# EPICS substitutions: EX2/scr/neurons_old.substitutions
file network.template {
	pattern { name, name-next, in1, w1, in2, w2, in3, w3, in4, w4}

		{ "11", "12-sum", "01", "01-11", "11", "11-11", "12", "12-11", "13", "13-11" }
		{ "12", "13-sum", "01", "01-12", "11", "11-12", "12", "12-12", "13", "13-12" }
		{ "13", "11-ac", "01", "01-13", "11", "11-13", "12", "12-13", "13", "13-13" }

		{ "21", "22-sum", "11", "11-21", "12", "12-21", "13", "13-21", "null", "null" }
		{ "22", "23-sum", "11", "11-22", "12", "12-22", "13", "13-22", "null", "null" }
		{ "23", "21-ac", "11", "11-23", "12", "12-23", "13", "13-23", "null", "null" }
}

file ac.template {
	pattern { name, name-next }
		{ "11", "12-ac" }
		{ "12", "13-ac" }
		{ "13", "21-sum" }

		{ "21", "22-ac" }
		{ "22", "23-ac" }
		{ "23", "score-fanout" }
}

file softmax.template {
	pattern { name, other1, other2 }
		{ "21", "22", "23" }
		{ "22", "21", "23" }
		{ "23", "21", "22" }
}

file weights.template {
	pattern { name1, name2, weight }
		{ "01", "11", "-50" }
		{ "01", "12", "1" }
		{ "01", "13", "50" }

		{ "11", "11", "0" }
		{ "12", "11", "50" }
		{ "13", "11", "0" }

		{ "11", "12", "0" }
		{ "12", "12", "0" }
		{ "13", "12", "0" }

		{ "11", "13", "0" }
		{ "12", "13", "-50" }
		{ "13", "13", "0" }

		{ "11", "21", "8" }
		{ "12", "21", "0" }
		{ "13", "21", "-8" }

		{ "11", "22", "-6" }
		{ "12", "22", "0" }
		{ "13", "22", "-6" }

		{ "11", "23", "-8" }
		{ "12", "23", "0" }
		{ "13", "23", "8" }
}

file bias.template {
	pattern { name, bias }

		{ "11", "-1" }
		{ "12", "0" }
		{ "13", "-1" }

		{ "21", "0" }
		{ "22", "3" }
		{ "23", "0" }
}
